FUNCTION Convert_SINT_TO_INT : Hresult
VAR_INPUT
	in : SINT;
	out : REFERENCE TO INT;
END_VAR
VAR
	converted : INT;
END_VAR

converted := SINT_TO_INT(in);

IF (INT_TO_SINT(converted) <> in) THEN
	Convert_SINT_TO_INT := INCOMPATIBLE;
	RETURN;
END_IF

out := converted;

END_FUNCTION

(* stored: Version 1.1.0.1, ProductVersion 3.1.4024.12
   POU Convert_SINT_TO_INT: Id {2813ceae-c54c-4785-8038-f135ae55f674}, SpecialFunc None *)
